# EPICS substitutions: ek9000App/Db/EL6002.substitutions
file EL6002.template
{       pattern
        {
                TERMINAL,

        }
        {
        }
}
